(* IEC 61131-3 sources: 83616---Application-of-Mechatronic-Systems---PROJECT/codesys_txt/Device.dev/Plc Logic/Application, 4 files *)

(* ---- typ_OrderData.dut ---- *)
(*#-#-#-#-#-#-#-#-#-#---Declaration---#-#-#-#-#-#-#-#-#-#-#-#-#*)

TYPE typ_OrderData :
STRUCT
	ulOrderNo: ULINT := 0;
	uiQty: DINT;
	eType: STRING;
	aeAccessories: ARRAY [1..4] OF STRING;
	status: STRING:='NA';
	asmLine: STRING:='NA';
END_STRUCT
END_TYPE

(* ---- typ_TypeStats.dut ---- *)
(*#-#-#-#-#-#-#-#-#-#---Declaration---#-#-#-#-#-#-#-#-#-#-#-#-#*)

TYPE typ_TypeStats :
STRUCT
	uiBMX:UINT;
	uiROAD:UINT;
	uiFOLDING:UINT;
	uiELECTRIC:UINT;
END_STRUCT
END_TYPE

(* ---- RAND.pou ---- *)
(*#-#-#-#-#-#-#-#-#-#---Declaration---#-#-#-#-#-#-#-#-#-#-#-#-#*)

FUNCTION_BLOCK RAND
VAR_INPUT
	IN_diMin: DINT;
	IN_diMax: DINT;
END_VAR
VAR_OUTPUT
	di_Result: DINT;
END_VAR
VAR
	di_Div: DINT;
	ARR: ARRAY [1..100] OF INT:=[3 ,  1  , 3  , 3  , 4  , 4  , 4  , 1 ,  1   ,2  , 3   ,4  , 3   ,1  , 4  , 3  , 3   ,2   ,1  , 4  , 4   ,3  , 1   ,2   ,1 ,2   ,3   ,3  , 3  , 1  , 3   ,4  , 4  , 3   ,2  , 4  , 2  , 4  , 4  , 1  , 2  , 2  , 4  , 2  , 2  , 4   ,4   ,1  , 4  , 2 ,2   ,1   ,3  , 3  , 3   ,4   ,2   ,4   ,3   ,1   ,1   ,4   ,3   ,1   ,2   ,4   ,1   ,4   ,2   ,1   ,2   ,4   ,1   ,2   ,1, 3   ,4   ,3   ,3   ,4   ,4   ,4   ,4   ,1   ,2   ,4   ,2   ,1   ,4   ,3  , 3   ,4   ,4   ,2   ,4   ,3   ,2   ,1   ,2   ,4];
END_VAR

(*#-#-#-#-#-#-#-#-#-#---Implementation---#-#-#-#-#-#-#-#-#-#-#-#-#*)

di_Div:=(IN_diMax-IN_diMin);
di_Result:=TO_DINT(SysTimeGetMs()) MOD (di_Div + 1);
di_Result:=ARR[di_Result];
//di_Result:=di_Result+IN_diMin;

(* ---- PLC_PRG.pou ---- *)
(*#-#-#-#-#-#-#-#-#-#---Declaration---#-#-#-#-#-#-#-#-#-#-#-#-#*)

PROGRAM PLC_PRG
VAR
fbWebServer:FB_WebServer;
fbAssemblyLine:ARRAY [0..4] OF FB_AssemblyLine;
fbAssemblyAdd: ARRAY[0..4] OF POINTER TO fb_AssemblyLine :=	[ADR(fbAssemblyLine[0]),
																 ADR(fbAssemblyLine[1]),
																 ADR(fbAssemblyLine[2]),
																 ADR(fbAssemblyLine[3]),
																 ADR(fbAssemblyLine[4])];
fbOrderParser: FB_OrderParser(pFB_Server := ADR(fbWebServer),apFB_AssemblyLine:=fbAssemblyAdd);
i:INT;
fb_Ass: FB_AssemblyLine;
assem_line:INT;
assembly_line: ARRAY [0..4] OF STRING:=['ASSEMBLY_LINE_1','ASSEMBLY_LINE_2','ASSEMBLY_LINE_3','ASSEMBLY_LINE_4','ASSEMBLY_LINE_5'];
Web_Visu: ARRAY [1..3] OF STRING:=['HMI_ORDER','Visu_Order','Visu_Assembly_Display'];
web: INT;
END_VAR
(*#-#-#-#-#-#-#-#-#-#---Implementation---#-#-#-#-#-#-#-#-#-#-#-#-#*)

fbWebServer(); //simulate web orders
fbOrderParser();
FOR I:=0 TO 4 BY 1 DO
	fbAssemblyLine[i]();
END_FOR
IF web=1 THEN
	CurrentVisu:='HMI_ORDER';
ELSIF web=2 THEN
	CurrentVisu:='Visu_Order';
ELSIF web=3 THEN
	CurrentVisu:='Visu_Assembly_Display';
END_IF
IF assem_line=0 THEN
	fb_Ass:=fbAssemblyLine[0];
ELSIF assem_line=1 THEN
	fb_Ass:=fbAssemblyLine[1];
ELSIF assem_line=2 THEN
	fb_Ass:=fbAssemblyLine[2];
ELSIF assem_line=3 THEN
	fb_Ass:=fbAssemblyLine[3];
ELSIF assem_line=4 THEN
	fb_Ass:=fbAssemblyLine[4];
END_IF
